Fanuc KAREL source: kx00009.KL

-- PROVISIONAL review KL for V940-1; original PC SHA256 6d08c3ae3eb55095c0a49ae01b567bdf34c1bb642a5b2672eab2acf5e7d9a7d7
-- Incomplete behavior may be omitted. Consult companion uncertainty JSON. Do not deploy.
PROGRAM KX00009
%NOLOCKGROUP
VAR
  I : INTEGER
  J : INTEGER
  B : BOOLEAN
  F : FILE
  S : STRING[80]
-- UNRESOLVED_DECL P type=000102
BEGIN
  -- V9_ZERO_TABLE_METADATA_HINT layout=0001; no indexed target words; source/name/runtime held
  -- UNRESOLVED_PC offsets 5-7; opcodes 9C,4F
  -- UNRESOLVED_PC offsets 12-16; opcodes 7F
END KX00009
